PROGRAM FAST
VAR
	fbTest:			FB_TestFast;
  	exception:			__SYSTEM.ExceptionCode;	
END_VAR

__TRY
	IF exception = __SYSTEM.ExceptionCode.RTSEXCPT_NOEXCEPTION THEN
		fbTest.P_Event.P_Logger:= MAIN.fbLogger;
	
	fbTest();
	
		
	END_IF


__CATCH(exception)


__ENDTRY

END_PROGRAM

(* stored: Version 1.1.0.1
   POU FAST: Id {56131508-6984-4602-9bc7-713829ff2f55}, SpecialFunc None *)
